PROGRAM Station1
VAR

END_VAR

END_PROGRAM

(* stored: Version 1.1.0.1
   POU Station1: Id {689f4e9b-42c0-4037-a3cd-3420e210bd57}, SpecialFunc None *)
